PROGRAM POU_TrendLine
VAR
	aiLoopIndex : DINT;
	ArrayTrend : ARRAY[1..GVL_Data.aiTrendArrayMax]OF REAL;
	ArrayTrendDisp : ARRAY[1..GVL_Data.aiTrendArrayMax]OF REAL;
END_VAR
VAR_INPUT
	rTrendlinePressure : LREAL;
END_VAR

// Trend array loop
FOR aiLoopIndex := 1 TO (GVL_Data.aiTrendArrayMax-1) DO
	ArrayTrend[aiLoopIndex] := ArrayTrend[aiLoopIndex + 1];
	
END_FOR

//ArrayTrend[GVL_Data.aiTrendArrayMax] := GVL_Data.fAnalogData;
ArrayTrend[GVL_Data.aiTrendArrayMax] := MAIN.fb_Gauge_01.rPressureTorr;

// When Pause is OFF, Update the ArrayTrendDisp Array
IF NOT GVL_Data.bTrendStatus THEN
	FOR aiLoopIndex := 1 TO GVL_Data.aiTrendArrayMax DO
		ArrayTrendDisp[aiLoopIndex] := ArrayTrend[aiLoopIndex + 1];
	END_FOR
END_IF

// Test code
GVL_Data.fTestDelta := 20.0;
IF GVL_Data.fAnalogData <= 980.0 THEN
	GVL_Data.fAnalogData := GVL_Data.fAnalogData + GVL_Data.fTestDelta;	
END_IF

IF GVL_Data.fAnalogData >= 1000.0 THEN
	GVL_Data.fAnalogData := 100.0;
END_IF

END_PROGRAM

(* stored: Version 1.1.0.1
   POU POU_TrendLine: Id {dfa9c779-5caa-46c4-91b7-45f046c2c72c}, SpecialFunc None *)
